PROGRAM POU_GetPosition
VAR
	fb_Axis1Position:MC_ReadActualPosition;
	fb_Axis2Position:MC_ReadActualPosition;
	fb_Axis3Position:MC_ReadActualPosition;
	fb_Axis4Position:MC_ReadActualPosition;
	fb_Axis5Position:MC_ReadActualPosition;
	fb_Axis6Position:MC_ReadActualPosition;
END_VAR

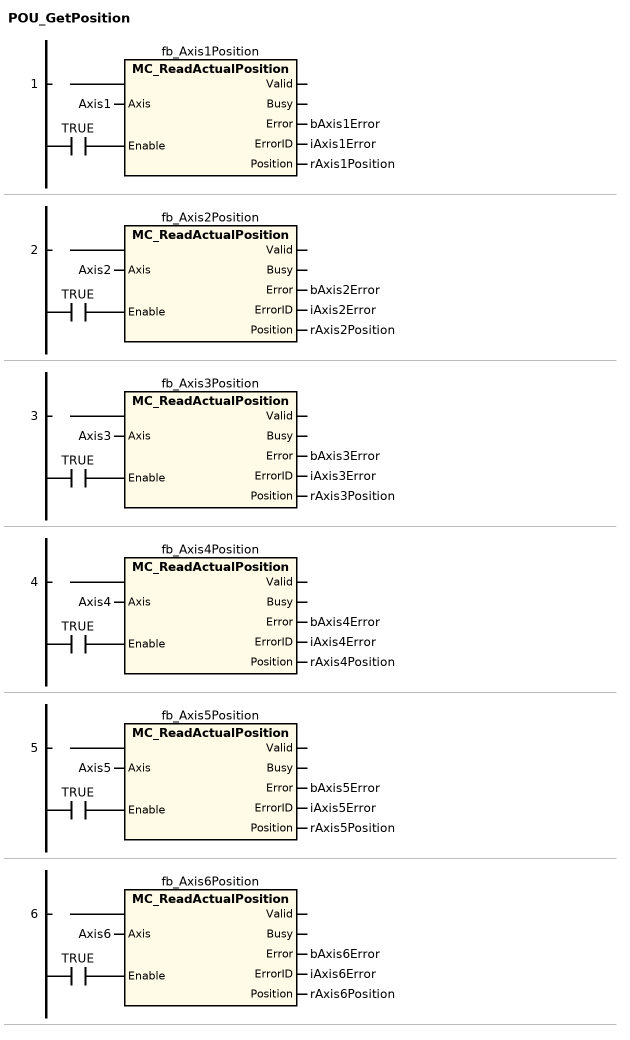
// NETWORK 1
fb_Axis1Position(
    Axis := Axis1,
    Enable := TRUE,
    Error => bAxis1Error,
    ErrorID => iAxis1Error,
    Position => rAxis1Position); // MC_ReadActualPosition

// NETWORK 2
fb_Axis2Position(
    Axis := Axis2,
    Enable := TRUE,
    Error => bAxis2Error,
    ErrorID => iAxis2Error,
    Position => rAxis2Position); // MC_ReadActualPosition

// NETWORK 3
fb_Axis3Position(
    Axis := Axis3,
    Enable := TRUE,
    Error => bAxis3Error,
    ErrorID => iAxis3Error,
    Position => rAxis3Position); // MC_ReadActualPosition

// NETWORK 4
fb_Axis4Position(
    Axis := Axis4,
    Enable := TRUE,
    Error => bAxis4Error,
    ErrorID => iAxis4Error,
    Position => rAxis4Position); // MC_ReadActualPosition

// NETWORK 5
fb_Axis5Position(
    Axis := Axis5,
    Enable := TRUE,
    Error => bAxis5Error,
    ErrorID => iAxis5Error,
    Position => rAxis5Position); // MC_ReadActualPosition

// NETWORK 6
fb_Axis6Position(
    Axis := Axis6,
    Enable := TRUE,
    Error => bAxis6Error,
    ErrorID => iAxis6Error,
    Position => rAxis6Position); // MC_ReadActualPosition

END_PROGRAM

(* stored: Version 1.1.0.1, ProductVersion 3.1.4022.18
   POU POU_GetPosition: Id {46d6defc-e8d7-4707-86d1-c2760a03dfb9}, SpecialFunc None *)
